{attribute 'qualified_only'}
{attribute 'strict'}
TYPE E_StewartState :
(
	TRANSIT := 0,
	OFF,
	SETTLED,
	OIL_HEATING,
	NEUTRAL,
	NEUTRAL_FREEZE,
	ENGAGED,
	ENGAGED_FREEZE	
) USINT;
END_TYPE

(* stored: Version 1.1.0.1, ProductVersion 3.1.4022.18
   DUT E_StewartState: Id {80c20507-7c0d-4412-8a64-b356b7316672} *)
